SYSTEM FactoryioLuaJITDemo
  (* Version 1.0, 2021-07-28, Tuojian Lyu *)
  APPLICATION VariablesInitApp
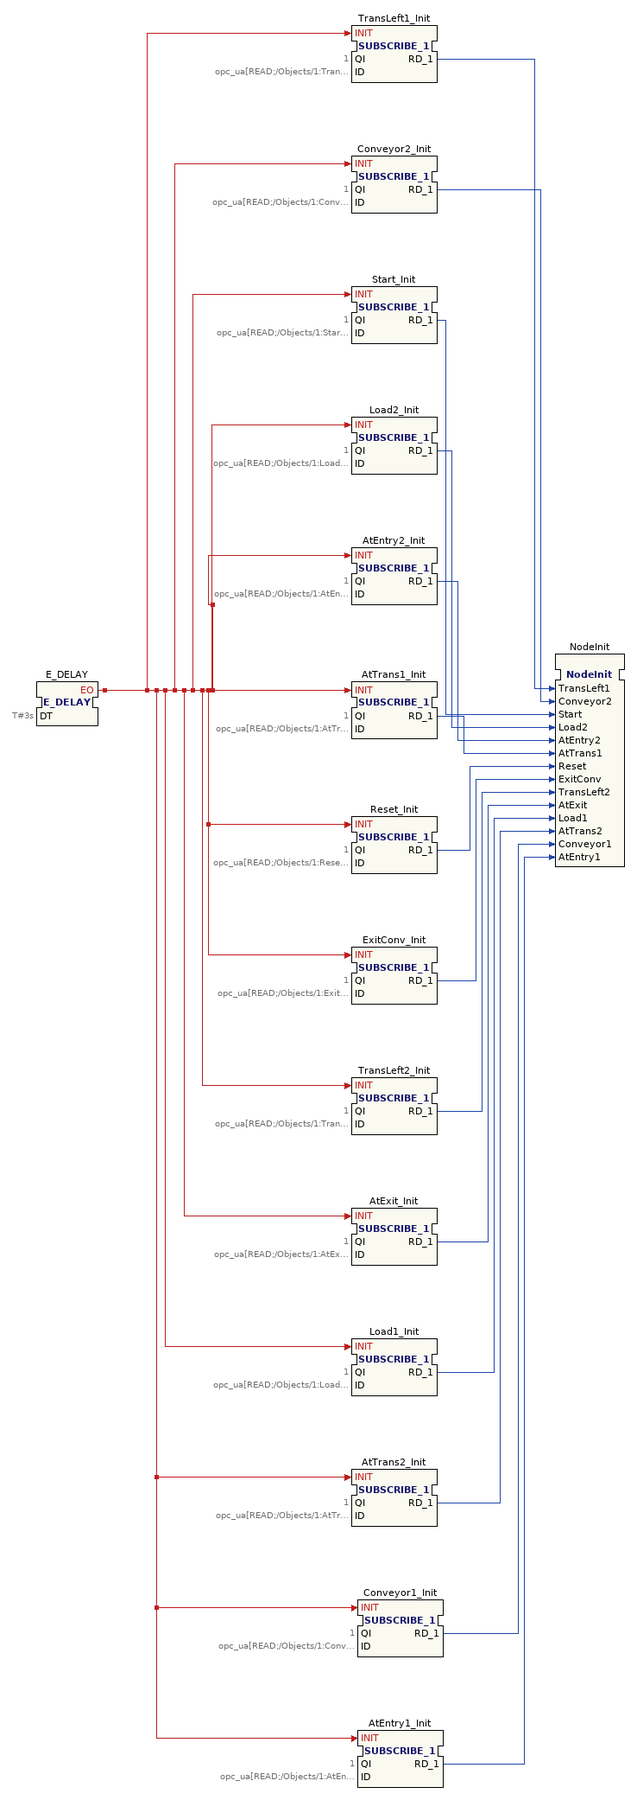
    FBS
      TransLeft1_Init : SUBSCRIBE_1(QI := 1, ID := opc_ua[READ;/Objects/1:TransLeft1]);
      Conveyor2_Init : SUBSCRIBE_1(QI := 1, ID := opc_ua[READ;/Objects/1:Conveyor2]);
      Start_Init : SUBSCRIBE_1(QI := 1, ID := opc_ua[READ;/Objects/1:Start]);
      AtEntry2_Init : SUBSCRIBE_1(QI := 1, ID := opc_ua[READ;/Objects/1:AtEntry2]);
      Load2_Init : SUBSCRIBE_1(QI := 1, ID := opc_ua[READ;/Objects/1:Load2]);
      Reset_Init : SUBSCRIBE_1(QI := 1, ID := opc_ua[READ;/Objects/1:Reset]);
      AtTrans1_Init : SUBSCRIBE_1(QI := 1, ID := opc_ua[READ;/Objects/1:AtTrans1]);
      TransLeft2_Init : SUBSCRIBE_1(QI := 1, ID := opc_ua[READ;/Objects/1:TransLeft2]);
      ExitConv_Init : SUBSCRIBE_1(QI := 1, ID := opc_ua[READ;/Objects/1:ExitConv]);
      Load1_Init : SUBSCRIBE_1(QI := 1, ID := opc_ua[READ;/Objects/1:Load1]);
      AtExit_Init : SUBSCRIBE_1(QI := 1, ID := opc_ua[READ;/Objects/1:AtExit]);
      AtTrans2_Init : SUBSCRIBE_1(QI := 1, ID := opc_ua[READ;/Objects/1:AtTrans2]);
      E_DELAY : E_DELAY(DT := T#3s);
      Conveyor1_Init : SUBSCRIBE_1(QI := 1, ID := opc_ua[READ;/Objects/1:Conveyor1]);
      AtEntry1_Init : SUBSCRIBE_1(QI := 1, ID := opc_ua[READ;/Objects/1:AtEntry1]);
      NodeInit : NodeInit;
    END_FBS
    EVENT_CONNECTIONS
      E_DELAY.EO TO TransLeft1_Init.INIT;
      E_DELAY.EO TO Conveyor2_Init.INIT;
      E_DELAY.EO TO Start_Init.INIT;
      E_DELAY.EO TO Load2_Init.INIT;
      E_DELAY.EO TO AtEntry2_Init.INIT;
      E_DELAY.EO TO AtTrans1_Init.INIT;
      E_DELAY.EO TO Reset_Init.INIT;
      E_DELAY.EO TO ExitConv_Init.INIT;
      E_DELAY.EO TO TransLeft2_Init.INIT;
      E_DELAY.EO TO AtExit_Init.INIT;
      E_DELAY.EO TO Load1_Init.INIT;
      E_DELAY.EO TO AtTrans2_Init.INIT;
      E_DELAY.EO TO Conveyor1_Init.INIT;
      E_DELAY.EO TO AtEntry1_Init.INIT;
    END_CONNECTIONS
    DATA_CONNECTIONS
      TransLeft1_Init.RD_1 TO NodeInit.TransLeft1;
      Conveyor2_Init.RD_1 TO NodeInit.Conveyor2;
      Start_Init.RD_1 TO NodeInit.Start;
      Load2_Init.RD_1 TO NodeInit.Load2;
      AtEntry2_Init.RD_1 TO NodeInit.AtEntry2;
      AtTrans1_Init.RD_1 TO NodeInit.AtTrans1;
      Reset_Init.RD_1 TO NodeInit.Reset;
      ExitConv_Init.RD_1 TO NodeInit.ExitConv;
      TransLeft2_Init.RD_1 TO NodeInit.TransLeft2;
      AtExit_Init.RD_1 TO NodeInit.AtExit;
      Load1_Init.RD_1 TO NodeInit.Load1;
      AtTrans2_Init.RD_1 TO NodeInit.AtTrans2;
      Conveyor1_Init.RD_1 TO NodeInit.Conveyor1;
      AtEntry1_Init.RD_1 TO NodeInit.AtEntry1;
    END_CONNECTIONS
  END_APPLICATION
  APPLICATION FactoryioLuaJITDemo
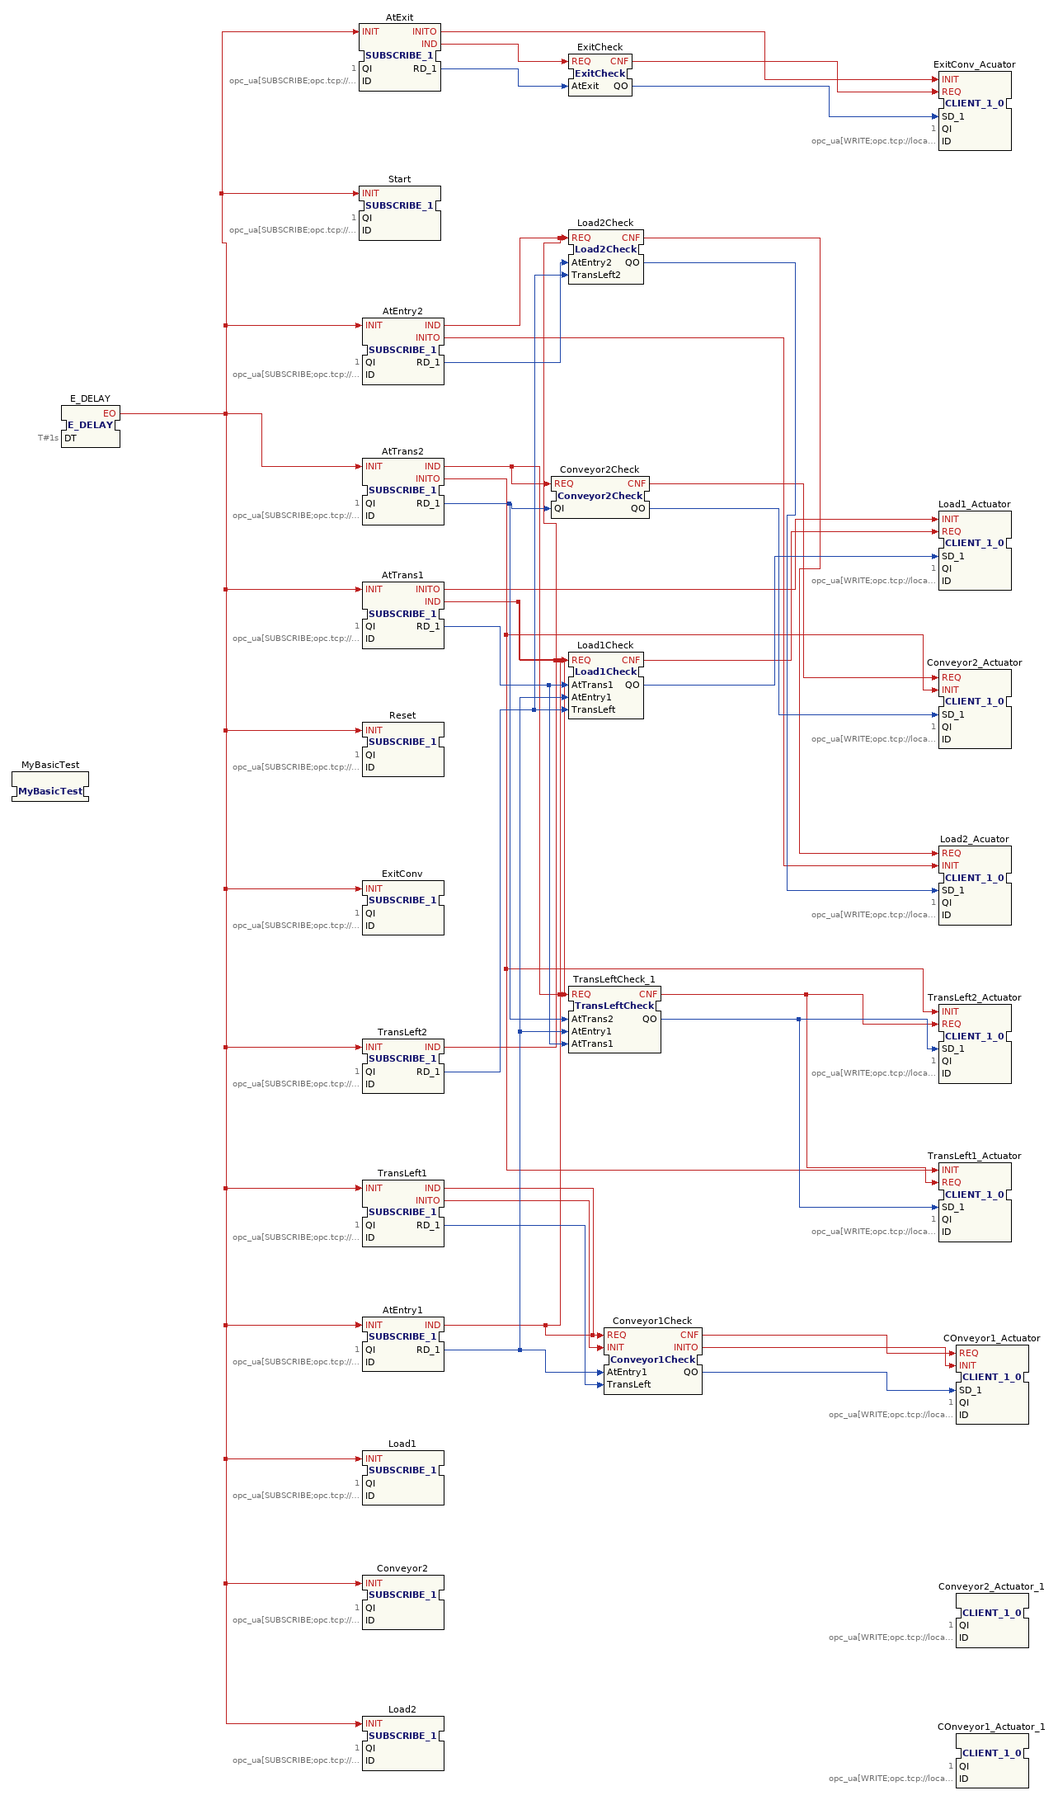
    FBS
      Load1_Actuator : CLIENT_1_0(QI := 1, ID := opc_ua[WRITE;opc.tcp://localhost:4840#;/Objects/1:Load1]);
      ExitConv_Acuator : CLIENT_1_0(QI := 1, ID := opc_ua[WRITE;opc.tcp://localhost:4840#;/Objects/1:ExitConv]);
      Start : SUBSCRIBE_1(QI := 1, ID := opc_ua[SUBSCRIBE;opc.tcp://localhost:4840#;/Objects/1:Start]);
      AtExit : SUBSCRIBE_1(QI := 1, ID := opc_ua[SUBSCRIBE;opc.tcp://localhost:4840#;/Objects/1:AtExit]);
      TransLeft1_Actuator : CLIENT_1_0(QI := 1, ID := opc_ua[WRITE;opc.tcp://localhost:4840#;/Objects/1:TransLeft1]);
      TransLeft2_Actuator : CLIENT_1_0(QI := 1, ID := opc_ua[WRITE;opc.tcp://localhost:4840#;/Objects/1:TransLeft2]);
      AtTrans2 : SUBSCRIBE_1(QI := 1, ID := opc_ua[SUBSCRIBE;opc.tcp://localhost:4840#;/Objects/1:AtTrans2]);
      Conveyor2_Actuator : CLIENT_1_0(QI := 1, ID := opc_ua[WRITE;opc.tcp://localhost:4840#;/Objects/1:Conveyor2]);
      AtEntry2 : SUBSCRIBE_1(QI := 1, ID := opc_ua[SUBSCRIBE;opc.tcp://localhost:4840#;/Objects/1:AtEntry2]);
      AtTrans1 : SUBSCRIBE_1(QI := 1, ID := opc_ua[SUBSCRIBE;opc.tcp://localhost:4840#;/Objects/1:AtTrans1]);
      E_DELAY : E_DELAY(DT := T#1s);
      ExitConv : SUBSCRIBE_1(QI := 1, ID := opc_ua[SUBSCRIBE;opc.tcp://localhost:4840#;/Objects/1:ExitConv]);
      Conveyor2 : SUBSCRIBE_1(QI := 1, ID := opc_ua[SUBSCRIBE;opc.tcp://localhost:4840#;/Objects/1:Conveyor2]);
      TransLeft2 : SUBSCRIBE_1(QI := 1, ID := opc_ua[SUBSCRIBE;opc.tcp://localhost:4840#;/Objects/1:TransLeft2]);
      Load1 : SUBSCRIBE_1(QI := 1, ID := opc_ua[SUBSCRIBE;opc.tcp://localhost:4840#;/Objects/1:Load1]);
      TransLeft1 : SUBSCRIBE_1(QI := 1, ID := opc_ua[SUBSCRIBE;opc.tcp://localhost:4840#;/Objects/1:TransLeft1]);
      Load2 : SUBSCRIBE_1(QI := 1, ID := opc_ua[SUBSCRIBE;opc.tcp://localhost:4840#;/Objects/1:Load2]);
      Reset : SUBSCRIBE_1(QI := 1, ID := opc_ua[SUBSCRIBE;opc.tcp://localhost:4840#;/Objects/1:Reset]);
      Load2_Acuator : CLIENT_1_0(QI := 1, ID := opc_ua[WRITE;opc.tcp://localhost:4840#;/Objects/1:Load2]);
      Conveyor2Check : Conveyor2Check;
      Load2Check : Load2Check;
      ExitCheck : ExitCheck;
      COnveyor1_Actuator : CLIENT_1_0(QI := 1, ID := opc_ua[WRITE;opc.tcp://localhost:4840#;/Objects/1:Conveyor1]);
      AtEntry1 : SUBSCRIBE_1(QI := 1, ID := opc_ua[SUBSCRIBE;opc.tcp://localhost:4840#;/Objects/1:AtEntry1]);
      Load1Check : Load1Check;
      Conveyor1Check : Conveyor1Check;
      TransLeftCheck_1 : TransLeftCheck;
      COnveyor1_Actuator_1 : CLIENT_1_0(QI := 1, ID := opc_ua[WRITE;opc.tcp://localhost:4840#;/Objects/1:Conveyor1]);
      Conveyor2_Actuator_1 : CLIENT_1_0(QI := 1, ID := opc_ua[WRITE;opc.tcp://localhost:4840#;/Objects/1:Conveyor2]);
      MyBasicTest : MyBasicTest;
    END_FBS
    EVENT_CONNECTIONS
      E_DELAY.EO TO AtExit.INIT;
      E_DELAY.EO TO Start.INIT;
      E_DELAY.EO TO AtEntry2.INIT;
      E_DELAY.EO TO AtTrans2.INIT;
      E_DELAY.EO TO AtTrans1.INIT;
      E_DELAY.EO TO TransLeft1.INIT;
      E_DELAY.EO TO ExitConv.INIT;
      E_DELAY.EO TO Load1.INIT;
      E_DELAY.EO TO Conveyor2.INIT;
      E_DELAY.EO TO TransLeft2.INIT;
      E_DELAY.EO TO Load2.INIT;
      E_DELAY.EO TO Reset.INIT;
      Conveyor2Check.CNF TO Conveyor2_Actuator.REQ;
      AtTrans2.IND TO Conveyor2Check.REQ;
      AtEntry2.IND TO Load2Check.REQ;
      Load2Check.CNF TO Load2_Acuator.REQ;
      AtTrans2.INITO TO Conveyor2_Actuator.INIT;
      AtEntry2.INITO TO Load2_Acuator.INIT;
      AtTrans2.INITO TO TransLeft2_Actuator.INIT;
      AtTrans2.INITO TO TransLeft1_Actuator.INIT;
      AtTrans1.INITO TO Load1_Actuator.INIT;
      AtExit.INITO TO ExitConv_Acuator.INIT;
      AtExit.IND TO ExitCheck.REQ;
      ExitCheck.CNF TO ExitConv_Acuator.REQ;
      E_DELAY.EO TO AtEntry1.INIT;
      AtTrans1.IND TO Load1Check.REQ;
      AtEntry1.IND TO Load1Check.REQ;
      TransLeft2.IND TO Load1Check.REQ;
      Load1Check.CNF TO Load1_Actuator.REQ;
      TransLeft2.IND TO Load2Check.REQ;
      AtEntry1.IND TO Conveyor1Check.REQ;
      TransLeft1.IND TO Conveyor1Check.REQ;
      Conveyor1Check.CNF TO COnveyor1_Actuator.REQ;
      TransLeft1.INITO TO Conveyor1Check.INIT;
      Conveyor1Check.INITO TO COnveyor1_Actuator.INIT;
      AtTrans2.IND TO TransLeftCheck_1.REQ;
      AtEntry1.IND TO TransLeftCheck_1.REQ;
      AtTrans1.IND TO TransLeftCheck_1.REQ;
      TransLeftCheck_1.CNF TO TransLeft2_Actuator.REQ;
      TransLeftCheck_1.CNF TO TransLeft1_Actuator.REQ;
    END_CONNECTIONS
    DATA_CONNECTIONS
      Conveyor2Check.QO TO Conveyor2_Actuator.SD_1;
      AtTrans2.RD_1 TO Conveyor2Check.QI;
      AtEntry2.RD_1 TO Load2Check.AtEntry2;
      TransLeft2.RD_1 TO Load2Check.TransLeft2;
      Load2Check.QO TO Load2_Acuator.SD_1;
      AtExit.RD_1 TO ExitCheck.AtExit;
      ExitCheck.QO TO ExitConv_Acuator.SD_1;
      AtTrans1.RD_1 TO Load1Check.AtTrans1;
      AtEntry1.RD_1 TO Load1Check.AtEntry1;
      TransLeft2.RD_1 TO Load1Check.TransLeft;
      Load1Check.QO TO Load1_Actuator.SD_1;
      AtEntry1.RD_1 TO Conveyor1Check.AtEntry1;
      TransLeft1.RD_1 TO Conveyor1Check.TransLeft;
      Conveyor1Check.QO TO COnveyor1_Actuator.SD_1;
      AtTrans2.RD_1 TO TransLeftCheck_1.AtTrans2;
      AtEntry1.RD_1 TO TransLeftCheck_1.AtEntry1;
      AtTrans1.RD_1 TO TransLeftCheck_1.AtTrans1;
      TransLeftCheck_1.QO TO TransLeft2_Actuator.SD_1;
      TransLeftCheck_1.QO TO TransLeft1_Actuator.SD_1;
    END_CONNECTIONS
  END_APPLICATION
  DEVICE FORTE_PC : FORTE_PC(MGR_ID := "localhost:61499")
    {SET_ATTRIBUTE(Profile, DynamicTypeLoad)} (* device profile *)
    {SET_ATTRIBUTE(FBType, GEN_E_MUX, F_LT, F_LWORD_TO_WORD, F_TAN, F_DINT_TO_UINT, F_BYTE_TO_DINT, F_ADD_DT_TIME, F_TIME_IN_US_TO_LREAL, F_INT_TO_UDINT, F_ADD_TOD_TIME, F_SUB_DT_DT, F_DT_TO_TOD, F_WSTRING_TO_REAL, F_UINT_TO_BCD_WORD, F_UDINT_TO_REAL, F_REAL_TO_UDINT, F_DWORD_TO_WORD, F_MUL, FB_CTUD_LINT, TEST_CONDITION, F_LE, GEN_SUBSCRIBE, F_LN, FB_CTD_DINT, GEN_OR, E_CYCLE, FB_F_TRIG, F_LREAL_TO_SINT, E_F_TRIG, F_LWORD_TO_UINT, E_RS, F_UINT_TO_WORD, F_WORD_TO_DINT, F_OR, F_WORD_TO_BYTE, F_TIME_IN_NS_TO_ULINT, FB_CTD_ULINT, FB_TOF, STEST_END, F_NE, FB_TON, F_STRING_TO_UINT, F_LWORD_TO_ULINT, F_INT_TO_STRING, F_INT_TO_BYTE, F_INT_TO_DINT, F_ULINT_TO_LINT, F_DWORD_TO_UINT, F_WSTRING_TO_ULINT, F_WSTRING_TO_LWORD, F_STRING_TO_DWORD, DWORD2DWORD, F_TIME_IN_NS_TO_LINT, F_DINT_TO_WSTRING, E_SELECT, F_LINT_TO_STRING, FB_CTUD, F_MULTIME, F_USINT_TO_INT, LocalizedText2LocalizedText, NodeInit, F_DWORD_TO_UDINT, F_UINT_TO_LWORD, F_SINT_TO_LWORD, GEN_F_MUX, USINT2USINT, F_LINT_TO_SINT, F_WORD_TO_USINT, F_DWORD_TO_INT, F_LREAL_TO_REAL, F_BOOL_TO_LINT, F_LEFT, FB_CTD, E_SR, F_UDINT_TO_BCD_DWORD, GEN_XOR, F_DINT_TO_WORD, F_SUB_TOD_TIME, E_RESTART, E_PERMIT, TIME2TIME, F_UINT_TO_SINT, F_XOR, F_STRING_TO_WORD, F_SEL, F_ULINT_TO_LREAL, F_SINT_TO_LREAL, F_DINT_TO_SINT, E_TimeOut, F_BYTE_TO_UDINT, F_REPLACE, F_LINT_TO_USINT, F_ABS, F_WORD_TO_LWORD, E_DELAY, GEN_ADD, F_INT_TO_WSTRING, F_STRING_TO_ULINT, F_USINT_TO_STRING, F_DINT_TO_USINT, F_STRING_TO_BOOL, F_DWORD_TO_WSTRING, F_INT_TO_REAL, F_DWORD_TO_STRING, E_CTU, F_TIME_TO_STRING, F_WSTRING_TO_BYTE, F_USINT_TO_WSTRING, F_WSTRING_TO_DINT, F_WSTRING_TO_DWORD, F_MOVE, F_WSTRING_TO_STRING, F_USINT_TO_LINT, F_DIV, F_WSTRING_TO_SINT, E_CTD, F_UINT_TO_DWORD, F_LWORD_TO_LINT, F_STRING_TO_TIME, FB_CTUD_DINT, F_ADD, F_BYTE_TO_LINT, F_TIME_IN_MS_TO_LREAL, F_LREAL_TO_UINT, F_ACOS, F_DWORD_TO_LINT, F_SHL, F_REAL_TO_ULINT, F_ULINT_TO_UINT, F_UDINT_TO_SINT, F_SHR, F_BOOL_TO_INT, UINT2UINT, F_WORD_TO_DWORD, F_INT_TO_LWORD, F_USINT_TO_UINT, F_LREAL_TO_WSTRING, F_INT_TO_ULINT, GEN_CSV_WRITER, F_LINT_TO_WORD, F_UINT_TO_LREAL, F_STRING_TO_SINT, F_SINT_TO_WORD, F_STRING_TO_WSTRING, STRING2STRING, F_LREAL_TO_DINT, F_SIN, F_UINT_TO_USINT, FB_CTU_LINT, F_DINT_TO_ULINT, F_REAL_TO_UINT, RMT_RES, F_ULINT_TO_WORD, F_INT_TO_LINT, E_D_FF, F_STRING_TO_USINT, FB_CTD_LINT, FB_R_TRIG, F_INT_TO_DWORD, F_WORD_TO_LINT, F_UDINT_TO_INT, REAL2REAL, F_LREAL_TO_STRING, F_WSTRING_TO_INT, F_LREAL_TO_USINT, F_DINT_TO_LWORD, DEV_MGR, F_SINT_TO_UINT, E_CTUD, E_RDELAY, F_SINT_TO_ULINT, F_LINT_TO_ULINT, F_RIGHT, F_SINT_TO_INT, F_LWORD_TO_WSTRING, SINT2SINT, FB_CTD_UDINT, F_LINT_TO_LWORD, F_LWORD_TO_UDINT, F_LWORD_TO_STRING, F_TRUNC, F_ULINT_TO_DWORD, F_TIME_IN_S_TO_LREAL, F_BOOL_TO_DWORD, E_TRAIN, OUT_ANY_CONSOLE, F_ULINT_TO_SINT, F_DINT_TO_LINT, F_BOOL_TO_USINT, F_UDINT_TO_DWORD, GEN_E_DEMUX, F_SQRT, F_BOOL_TO_DINT, F_BOOL_TO_BYTE, F_UINT_TO_INT, F_TIME_IN_S_TO_LINT, F_ULINT_TO_USINT, F_UINT_TO_REAL, F_LREAL_TO_LWORD, F_SINT_TO_LINT, F_MAX, F_LREAL_TO_INT, F_UDINT_TO_LWORD, INT2INT, F_BYTE_TO_ULINT, F_UDINT_TO_WORD, F_LINT_TO_UINT, F_TIME_IN_US_TO_ULINT, F_COS, F_TIME_IN_NS_TO_LREAL, F_REAL_TO_LINT, F_STRING_TO_LWORD, F_BYTE_TO_STRING, F_USINT_TO_WORD, E_REND, F_ASIN, F_REAL_TO_INT, F_BOOL_TO_LWORD, F_WORD_BCD_TO_UINT, F_BOOL_TO_SINT, F_BYTE_TO_INT, F_BOOL_TO_ULINT, EMB_RES, F_BYTE_TO_WORD, F_STRING_TO_INT, F_USINT_TO_LWORD, F_DWORD_TO_DINT, F_ULINT_TO_LWORD, GEN_APPEND_STRING, F_USINT_TO_ULINT, GEN_SUBL, F_DWORD_TO_BYTE, F_DIVTIME, F_ROL, F_LWORD_TO_DINT, F_WORD_TO_SINT, F_STRING_TO_REAL, F_LWORD_TO_BYTE, FB_CTU_DINT, GEN_AND, F_AND, F_ROR, GEN_CLIENT, F_ULINT_TO_WSTRING, F_SINT_TO_STRING, F_LREAL_TO_LINT, WSTRING2WSTRING, F_WORD_TO_INT, F_UINT_TO_BYTE, F_UDINT_TO_UINT, F_SINT_TO_UDINT, F_UINT_TO_DINT, F_UINT_TO_UDINT, F_UINT_TO_WSTRING, F_WSTRING_TO_UINT, F_DINT_TO_UDINT, E_SPLIT, F_DWORD_TO_LWORD, F_USINT_TO_SINT, F_ULINT_TO_BCD_LWORD, F_BYTE_BCD_TO_USINT, F_DWORD_TO_ULINT, F_BYTE_TO_SINT, F_BYTE_TO_WSTRING, GEN_ARRAY2ARRAY, F_DT_TO_DATE, GEN_STRUCT_DEMUX, F_LEN, GEN_STRUCT_MUX, F_INT_TO_WORD, FB_RANDOM, F_LINT_TO_UDINT, F_EXP, F_USINT_TO_DWORD, F_TIME_IN_MS_TO_ULINT, F_REAL_TO_SINT, F_INT_TO_USINT, F_UDINT_TO_WSTRING, F_EXPT, F_SUB, F_ULINT_TO_REAL, F_REAL_TO_LREAL, F_MID, F_BYTE_TO_UINT, F_BYTE_TO_DWORD, F_INT_TO_UINT, F_DWORD_TO_REAL, F_DINT_TO_BYTE, F_WORD_TO_STRING, F_REAL_TO_STRING, F_SUB_TOD_TOD, SET_AT_INDEX, F_MIN, F_LREAL_TO_ULINT, F_STRING_TO_BYTE, F_BYTE_TO_LWORD, F_STRING_TO_DINT, F_WORD_TO_WSTRING, BOOL2BOOL, F_LINT_TO_INT, F_WSTRING_TO_TIME, FB_CTU_UDINT, F_WSTRING_TO_BOOL, F_INSERT, F_SUB_DT_TIME, F_FIND, F_UDINT_TO_ULINT, F_WORD_TO_UDINT, F_DINT_TO_DWORD, F_WSTRING_TO_USINT, GEN_VALUES2ARRAY, GEN_ARRAY2VALUES, F_WSTRING_TO_WORD, F_DINT_TO_STRING, F_WORD_TO_UINT, F_TIME_IN_US_TO_LINT, F_LINT_TO_DWORD, F_CONCAT, FB_CTUD_ULINT, F_UDINT_TO_LINT, F_SUB_DATE_DATE, F_LWORD_TO_LREAL, F_LWORD_TO_INT, WORD2WORD, E_STOPWATCH, F_LIMIT, F_TIME_IN_S_TO_ULINT, F_LWORD_TO_USINT, F_REAL_TO_DINT, F_DWORD_TO_USINT, E_MERGE, F_SINT_TO_DWORD, E_DEMUX, F_BOOL_TO_UDINT, BYTE2BYTE, FB_TP, F_USINT_TO_BCD_BYTE, F_SINT_TO_DINT, F_UINT_TO_LINT, F_SINT_TO_BYTE, F_ATAN, F_LINT_TO_BYTE, F_BYTE_TO_USINT, F_ULINT_TO_UDINT, FB_SR, F_NOT, F_DINT_TO_INT, F_LINT_TO_DINT, F_DELETE, FB_CTU, GEN_SERVER, GEN_PUBL, F_UDINT_TO_LREAL, F_BOOL_TO_UINT, F_UINT_TO_STRING, E_R_TRIG, F_GE, F_LWORD_BCD_TO_ULINT, F_UDINT_TO_STRING, F_REAL_TO_WSTRING, FB_RS, F_MUX_2, F_LINT_TO_WSTRING, F_USINT_TO_UDINT, F_UINT_TO_ULINT, F_EQ, E_T_FF, F_USINT_TO_REAL, LREAL2LREAL, F_STRING_TO_LREAL, F_ULINT_TO_STRING, F_MOD, E_RTimeOut, F_ULINT_TO_DINT, F_ULINT_TO_BYTE, F_WSTRING_TO_UDINT, F_TIME_TO_WSTRING, GET_STRUCT_VALUE, GEN_PUBLISH, F_REAL_TO_DWORD, F_DWORD_BCD_TO_UDINT, F_INT_TO_LREAL, F_SINT_TO_WSTRING, F_LWORD_TO_SINT, F_GT, F_LINT_TO_REAL, F_TIME_IN_MS_TO_LINT, F_SINT_TO_REAL, F_LOG, F_ULINT_TO_INT, F_DWORD_TO_SINT, F_BOOL_TO_WORD, F_REAL_TO_USINT, E_SWITCH, F_LINT_TO_LREAL, F_STRING_TO_LINT, F_SINT_TO_USINT, F_DINT_TO_REAL, DINT2DINT, F_WORD_TO_ULINT, F_INT_TO_SINT, F_CONCAT_DATE_TOD, F_WSTRING_TO_LREAL, GET_AT_INDEX, F_USINT_TO_LREAL, F_BOOL_TO_WSTRING, FB_CTU_ULINT, F_DINT_TO_LREAL, UDINT2UDINT, F_USINT_TO_BYTE, F_BOOL_TO_STRING, F_LWORD_TO_DWORD, F_LREAL_TO_UDINT, F_STRING_TO_UDINT, F_UDINT_TO_DINT, F_UDINT_TO_BYTE, F_WSTRING_TO_LINT, F_USINT_TO_DINT)} (* created during deployment *)
    RESOURCE EMB_RES : EMB_RES
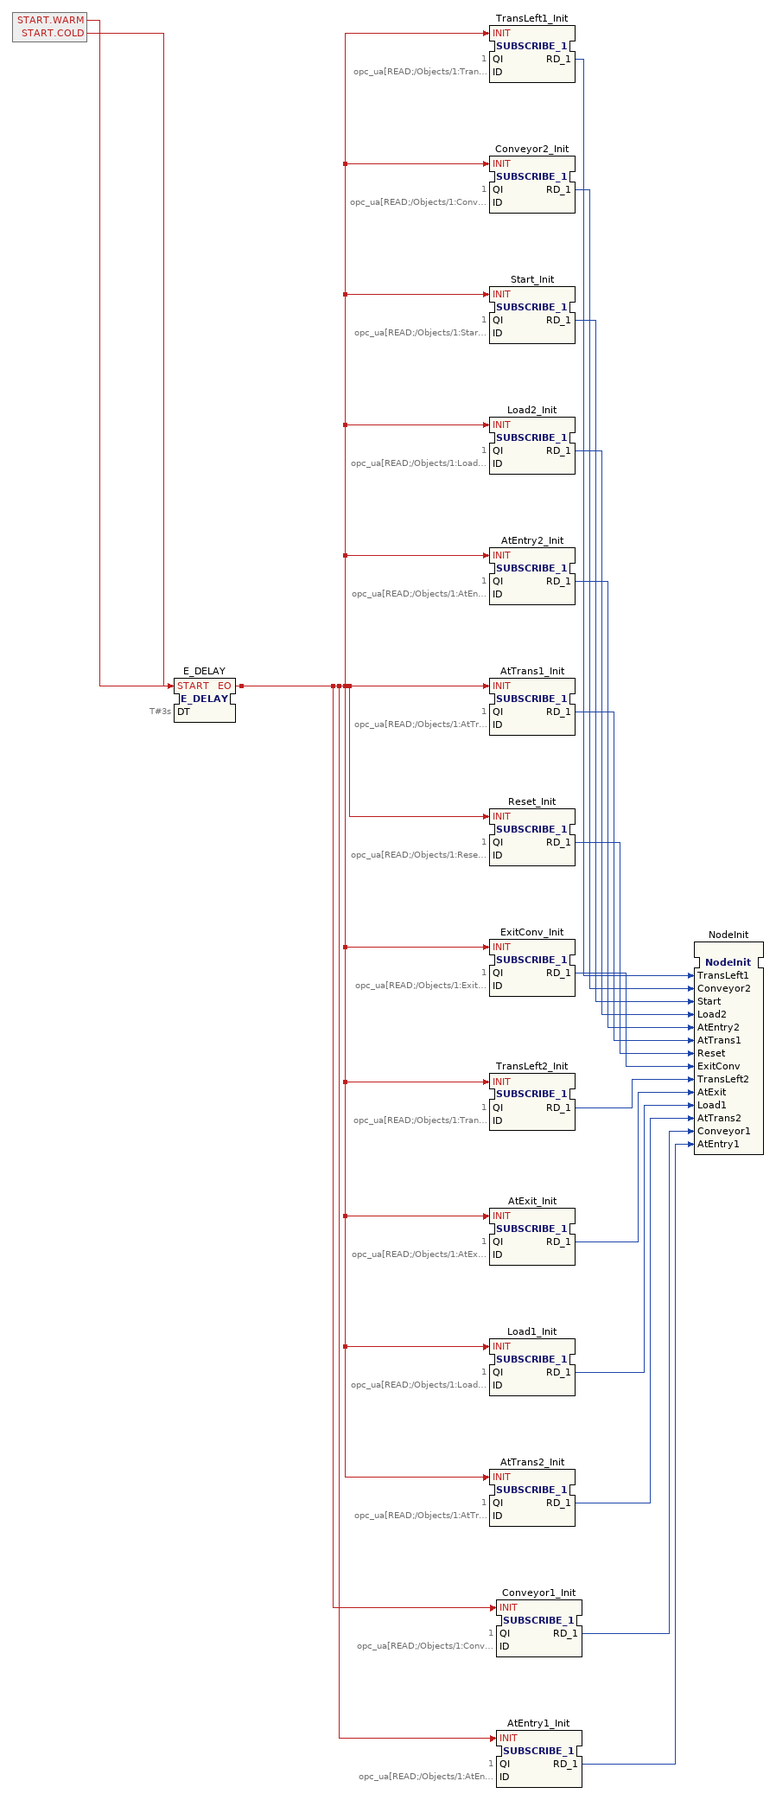
      FBS
        E_DELAY : E_DELAY(DT := T#3s);
        AtTrans2_Init : SUBSCRIBE_1(QI := 1, ID := opc_ua[READ;/Objects/1:AtTrans2]);
        AtExit_Init : SUBSCRIBE_1(QI := 1, ID := opc_ua[READ;/Objects/1:AtExit]);
        Load1_Init : SUBSCRIBE_1(QI := 1, ID := opc_ua[READ;/Objects/1:Load1]);
        ExitConv_Init : SUBSCRIBE_1(QI := 1, ID := opc_ua[READ;/Objects/1:ExitConv]);
        TransLeft2_Init : SUBSCRIBE_1(QI := 1, ID := opc_ua[READ;/Objects/1:TransLeft2]);
        AtTrans1_Init : SUBSCRIBE_1(QI := 1, ID := opc_ua[READ;/Objects/1:AtTrans1]);
        Reset_Init : SUBSCRIBE_1(QI := 1, ID := opc_ua[READ;/Objects/1:Reset]);
        Load2_Init : SUBSCRIBE_1(QI := 1, ID := opc_ua[READ;/Objects/1:Load2]);
        AtEntry2_Init : SUBSCRIBE_1(QI := 1, ID := opc_ua[READ;/Objects/1:AtEntry2]);
        Start_Init : SUBSCRIBE_1(QI := 1, ID := opc_ua[READ;/Objects/1:Start]);
        Conveyor2_Init : SUBSCRIBE_1(QI := 1, ID := opc_ua[READ;/Objects/1:Conveyor2]);
        TransLeft1_Init : SUBSCRIBE_1(QI := 1, ID := opc_ua[READ;/Objects/1:TransLeft1]);
        Conveyor1_Init : SUBSCRIBE_1(QI := 1, ID := opc_ua[READ;/Objects/1:Conveyor1]);
        AtEntry1_Init : SUBSCRIBE_1(QI := 1, ID := opc_ua[READ;/Objects/1:AtEntry1]);
        NodeInit : NodeInit;
      END_FBS
      EVENT_CONNECTIONS
        START.WARM TO E_DELAY.START;
        START.COLD TO E_DELAY.START;
        E_DELAY.EO TO AtTrans2_Init.INIT;
        E_DELAY.EO TO AtExit_Init.INIT;
        E_DELAY.EO TO Load1_Init.INIT;
        E_DELAY.EO TO ExitConv_Init.INIT;
        E_DELAY.EO TO TransLeft2_Init.INIT;
        E_DELAY.EO TO AtTrans1_Init.INIT;
        E_DELAY.EO TO Reset_Init.INIT;
        E_DELAY.EO TO Load2_Init.INIT;
        E_DELAY.EO TO AtEntry2_Init.INIT;
        E_DELAY.EO TO Start_Init.INIT;
        E_DELAY.EO TO Conveyor2_Init.INIT;
        E_DELAY.EO TO TransLeft1_Init.INIT;
        E_DELAY.EO TO Conveyor1_Init.INIT;
        E_DELAY.EO TO AtEntry1_Init.INIT;
      END_CONNECTIONS
      DATA_CONNECTIONS
        TransLeft1_Init.RD_1 TO NodeInit.TransLeft1;
        Conveyor2_Init.RD_1 TO NodeInit.Conveyor2;
        Start_Init.RD_1 TO NodeInit.Start;
        Load2_Init.RD_1 TO NodeInit.Load2;
        AtEntry2_Init.RD_1 TO NodeInit.AtEntry2;
        AtTrans1_Init.RD_1 TO NodeInit.AtTrans1;
        Reset_Init.RD_1 TO NodeInit.Reset;
        ExitConv_Init.RD_1 TO NodeInit.ExitConv;
        TransLeft2_Init.RD_1 TO NodeInit.TransLeft2;
        AtExit_Init.RD_1 TO NodeInit.AtExit;
        Load1_Init.RD_1 TO NodeInit.Load1;
        AtTrans2_Init.RD_1 TO NodeInit.AtTrans2;
        Conveyor1_Init.RD_1 TO NodeInit.Conveyor1;
        AtEntry1_Init.RD_1 TO NodeInit.AtEntry1;
      END_CONNECTIONS
    END_RESOURCE
  END_DEVICE
  DEVICE FORTE_PC_1 : FORTE_PC(MGR_ID := "localhost:61500")
    {SET_ATTRIBUTE(Profile, DynamicTypeLoad)} (* device profile *)
    {SET_ATTRIBUTE(FBType, GEN_E_MUX, F_LT, F_LWORD_TO_WORD, F_TAN, F_DINT_TO_UINT, F_BYTE_TO_DINT, F_ADD_DT_TIME, F_TIME_IN_US_TO_LREAL, F_INT_TO_UDINT, F_ADD_TOD_TIME, F_SUB_DT_DT, F_DT_TO_TOD, F_WSTRING_TO_REAL, F_UINT_TO_BCD_WORD, F_UDINT_TO_REAL, F_REAL_TO_UDINT, F_DWORD_TO_WORD, F_MUL, FB_CTUD_LINT, TEST_CONDITION, F_LE, GEN_SUBSCRIBE, F_LN, FB_CTD_DINT, GEN_OR, E_CYCLE, FB_F_TRIG, F_LREAL_TO_SINT, E_F_TRIG, F_LWORD_TO_UINT, E_RS, F_UINT_TO_WORD, F_WORD_TO_DINT, F_OR, F_WORD_TO_BYTE, F_TIME_IN_NS_TO_ULINT, FB_CTD_ULINT, FB_TOF, STEST_END, F_NE, FB_TON, F_STRING_TO_UINT, F_LWORD_TO_ULINT, F_INT_TO_STRING, F_INT_TO_BYTE, F_INT_TO_DINT, F_ULINT_TO_LINT, F_DWORD_TO_UINT, F_WSTRING_TO_ULINT, F_WSTRING_TO_LWORD, F_STRING_TO_DWORD, DWORD2DWORD, F_TIME_IN_NS_TO_LINT, F_DINT_TO_WSTRING, E_SELECT, F_LINT_TO_STRING, FB_CTUD, F_MULTIME, F_USINT_TO_INT, LocalizedText2LocalizedText, F_DWORD_TO_UDINT, F_UINT_TO_LWORD, F_SINT_TO_LWORD, GEN_F_MUX, USINT2USINT, F_LINT_TO_SINT, F_WORD_TO_USINT, F_DWORD_TO_INT, F_LREAL_TO_REAL, F_BOOL_TO_LINT, F_LEFT, FB_CTD, E_SR, F_UDINT_TO_BCD_DWORD, GEN_XOR, F_DINT_TO_WORD, F_SUB_TOD_TIME, E_RESTART, E_PERMIT, TIME2TIME, F_UINT_TO_SINT, F_XOR, F_STRING_TO_WORD, F_SEL, F_ULINT_TO_LREAL, F_SINT_TO_LREAL, F_DINT_TO_SINT, E_TimeOut, F_BYTE_TO_UDINT, F_REPLACE, F_LINT_TO_USINT, F_ABS, F_WORD_TO_LWORD, MyBasicTest, E_DELAY, GEN_ADD, F_INT_TO_WSTRING, F_STRING_TO_ULINT, F_USINT_TO_STRING, F_DINT_TO_USINT, F_STRING_TO_BOOL, F_DWORD_TO_WSTRING, F_INT_TO_REAL, F_DWORD_TO_STRING, E_CTU, F_TIME_TO_STRING, F_WSTRING_TO_BYTE, F_USINT_TO_WSTRING, F_WSTRING_TO_DINT, F_WSTRING_TO_DWORD, F_MOVE, F_WSTRING_TO_STRING, F_USINT_TO_LINT, F_DIV, F_WSTRING_TO_SINT, E_CTD, F_UINT_TO_DWORD, F_LWORD_TO_LINT, F_STRING_TO_TIME, FB_CTUD_DINT, F_ADD, F_BYTE_TO_LINT, F_TIME_IN_MS_TO_LREAL, F_LREAL_TO_UINT, F_ACOS, F_DWORD_TO_LINT, F_SHL, F_REAL_TO_ULINT, F_ULINT_TO_UINT, F_UDINT_TO_SINT, F_SHR, F_BOOL_TO_INT, UINT2UINT, F_WORD_TO_DWORD, F_INT_TO_LWORD, F_USINT_TO_UINT, F_LREAL_TO_WSTRING, F_INT_TO_ULINT, GEN_CSV_WRITER, F_LINT_TO_WORD, F_UINT_TO_LREAL, F_STRING_TO_SINT, F_SINT_TO_WORD, F_STRING_TO_WSTRING, STRING2STRING, F_LREAL_TO_DINT, F_SIN, F_UINT_TO_USINT, FB_CTU_LINT, F_DINT_TO_ULINT, F_REAL_TO_UINT, RMT_RES, F_ULINT_TO_WORD, F_INT_TO_LINT, E_D_FF, F_STRING_TO_USINT, FB_CTD_LINT, FB_R_TRIG, F_INT_TO_DWORD, F_WORD_TO_LINT, F_UDINT_TO_INT, REAL2REAL, F_LREAL_TO_STRING, F_WSTRING_TO_INT, F_LREAL_TO_USINT, F_DINT_TO_LWORD, DEV_MGR, F_SINT_TO_UINT, E_CTUD, E_RDELAY, F_SINT_TO_ULINT, F_LINT_TO_ULINT, F_RIGHT, F_SINT_TO_INT, F_LWORD_TO_WSTRING, SINT2SINT, FB_CTD_UDINT, F_LINT_TO_LWORD, F_LWORD_TO_UDINT, F_LWORD_TO_STRING, F_TRUNC, F_ULINT_TO_DWORD, F_TIME_IN_S_TO_LREAL, F_BOOL_TO_DWORD, E_TRAIN, OUT_ANY_CONSOLE, F_ULINT_TO_SINT, F_DINT_TO_LINT, F_BOOL_TO_USINT, F_UDINT_TO_DWORD, GEN_E_DEMUX, F_SQRT, F_BOOL_TO_DINT, F_BOOL_TO_BYTE, F_UINT_TO_INT, F_TIME_IN_S_TO_LINT, F_ULINT_TO_USINT, F_UINT_TO_REAL, F_LREAL_TO_LWORD, F_SINT_TO_LINT, F_MAX, F_LREAL_TO_INT, F_UDINT_TO_LWORD, INT2INT, F_BYTE_TO_ULINT, F_UDINT_TO_WORD, F_LINT_TO_UINT, F_TIME_IN_US_TO_ULINT, F_COS, Conveyor2Check, F_TIME_IN_NS_TO_LREAL, F_REAL_TO_LINT, F_STRING_TO_LWORD, F_BYTE_TO_STRING, F_USINT_TO_WORD, E_REND, F_ASIN, TransLeftCheck, F_REAL_TO_INT, F_BOOL_TO_LWORD, F_WORD_BCD_TO_UINT, F_BOOL_TO_SINT, F_BYTE_TO_INT, F_BOOL_TO_ULINT, EMB_RES, F_BYTE_TO_WORD, F_STRING_TO_INT, F_USINT_TO_LWORD, F_DWORD_TO_DINT, F_ULINT_TO_LWORD, GEN_APPEND_STRING, F_USINT_TO_ULINT, GEN_SUBL, F_DWORD_TO_BYTE, F_DIVTIME, ExitCheck, F_ROL, F_LWORD_TO_DINT, F_WORD_TO_SINT, F_STRING_TO_REAL, F_LWORD_TO_BYTE, FB_CTU_DINT, GEN_AND, F_AND, F_ROR, GEN_CLIENT, F_ULINT_TO_WSTRING, F_SINT_TO_STRING, F_LREAL_TO_LINT, WSTRING2WSTRING, F_WORD_TO_INT, F_UINT_TO_BYTE, F_UDINT_TO_UINT, F_SINT_TO_UDINT, F_UINT_TO_DINT, F_UINT_TO_UDINT, F_UINT_TO_WSTRING, F_WSTRING_TO_UINT, F_DINT_TO_UDINT, E_SPLIT, F_DWORD_TO_LWORD, F_USINT_TO_SINT, F_ULINT_TO_BCD_LWORD, F_BYTE_BCD_TO_USINT, F_DWORD_TO_ULINT, F_BYTE_TO_SINT, F_BYTE_TO_WSTRING, GEN_ARRAY2ARRAY, F_DT_TO_DATE, GEN_STRUCT_DEMUX, F_LEN, GEN_STRUCT_MUX, F_INT_TO_WORD, FB_RANDOM, F_LINT_TO_UDINT, F_EXP, F_USINT_TO_DWORD, F_TIME_IN_MS_TO_ULINT, F_REAL_TO_SINT, F_INT_TO_USINT, Load2Check, F_UDINT_TO_WSTRING, F_EXPT, F_SUB, F_ULINT_TO_REAL, F_REAL_TO_LREAL, F_MID, F_BYTE_TO_UINT, F_BYTE_TO_DWORD, F_INT_TO_UINT, F_DWORD_TO_REAL, F_DINT_TO_BYTE, F_WORD_TO_STRING, F_REAL_TO_STRING, F_SUB_TOD_TOD, SET_AT_INDEX, F_MIN, F_LREAL_TO_ULINT, F_STRING_TO_BYTE, F_BYTE_TO_LWORD, F_STRING_TO_DINT, F_WORD_TO_WSTRING, BOOL2BOOL, F_LINT_TO_INT, F_WSTRING_TO_TIME, FB_CTU_UDINT, F_WSTRING_TO_BOOL, F_INSERT, F_SUB_DT_TIME, F_FIND, F_UDINT_TO_ULINT, F_WORD_TO_UDINT, F_DINT_TO_DWORD, Load1Check, F_WSTRING_TO_USINT, GEN_VALUES2ARRAY, GEN_ARRAY2VALUES, F_WSTRING_TO_WORD, F_DINT_TO_STRING, F_WORD_TO_UINT, F_TIME_IN_US_TO_LINT, F_LINT_TO_DWORD, F_CONCAT, FB_CTUD_ULINT, F_UDINT_TO_LINT, F_SUB_DATE_DATE, F_LWORD_TO_LREAL, F_LWORD_TO_INT, WORD2WORD, E_STOPWATCH, F_LIMIT, F_TIME_IN_S_TO_ULINT, F_LWORD_TO_USINT, F_REAL_TO_DINT, F_DWORD_TO_USINT, E_MERGE, F_SINT_TO_DWORD, E_DEMUX, F_BOOL_TO_UDINT, BYTE2BYTE, FB_TP, F_USINT_TO_BCD_BYTE, F_SINT_TO_DINT, F_UINT_TO_LINT, F_SINT_TO_BYTE, F_ATAN, F_LINT_TO_BYTE, F_BYTE_TO_USINT, F_ULINT_TO_UDINT, FB_SR, F_NOT, F_DINT_TO_INT, F_LINT_TO_DINT, F_DELETE, FB_CTU, GEN_SERVER, GEN_PUBL, F_UDINT_TO_LREAL, F_BOOL_TO_UINT, F_UINT_TO_STRING, E_R_TRIG, F_GE, F_LWORD_BCD_TO_ULINT, F_UDINT_TO_STRING, F_REAL_TO_WSTRING, FB_RS, F_MUX_2, F_LINT_TO_WSTRING, F_USINT_TO_UDINT, F_UINT_TO_ULINT, F_EQ, E_T_FF, F_USINT_TO_REAL, LREAL2LREAL, F_STRING_TO_LREAL, F_ULINT_TO_STRING, F_MOD, E_RTimeOut, F_ULINT_TO_DINT, F_ULINT_TO_BYTE, F_WSTRING_TO_UDINT, F_TIME_TO_WSTRING, GET_STRUCT_VALUE, GEN_PUBLISH, F_REAL_TO_DWORD, F_DWORD_BCD_TO_UDINT, F_INT_TO_LREAL, F_SINT_TO_WSTRING, Conveyor1Check, F_LWORD_TO_SINT, F_GT, F_LINT_TO_REAL, F_TIME_IN_MS_TO_LINT, F_SINT_TO_REAL, F_LOG, F_ULINT_TO_INT, F_DWORD_TO_SINT, F_BOOL_TO_WORD, F_REAL_TO_USINT, E_SWITCH, F_LINT_TO_LREAL, F_STRING_TO_LINT, F_SINT_TO_USINT, F_DINT_TO_REAL, DINT2DINT, F_WORD_TO_ULINT, F_INT_TO_SINT, F_CONCAT_DATE_TOD, F_WSTRING_TO_LREAL, GET_AT_INDEX, F_USINT_TO_LREAL, F_BOOL_TO_WSTRING, FB_CTU_ULINT, F_DINT_TO_LREAL, UDINT2UDINT, F_USINT_TO_BYTE, F_BOOL_TO_STRING, F_LWORD_TO_DWORD, F_LREAL_TO_UDINT, F_STRING_TO_UDINT, F_UDINT_TO_DINT, F_UDINT_TO_BYTE, F_WSTRING_TO_LINT, F_USINT_TO_DINT)} (* created during deployment *)
    RESOURCE EMB_RES : EMB_RES
      FBS
        TransLeftCheck_1 : TransLeftCheck;
        Conveyor1Check : Conveyor1Check;
        Load1Check : Load1Check;
        AtEntry1 : SUBSCRIBE_1(QI := 1, ID := opc_ua[SUBSCRIBE;opc.tcp://localhost:4840#;/Objects/1:AtEntry1]);
        COnveyor1_Actuator : CLIENT_1_0(QI := 1, ID := opc_ua[WRITE;opc.tcp://localhost:4840#;/Objects/1:Conveyor1]);
        ExitCheck : ExitCheck;
        Load2Check : Load2Check;
        Conveyor2Check : Conveyor2Check;
        Load2_Acuator : CLIENT_1_0(QI := 1, ID := opc_ua[WRITE;opc.tcp://localhost:4840#;/Objects/1:Load2]);
        Reset : SUBSCRIBE_1(QI := 1, ID := opc_ua[SUBSCRIBE;opc.tcp://localhost:4840#;/Objects/1:Reset]);
        Load2 : SUBSCRIBE_1(QI := 1, ID := opc_ua[SUBSCRIBE;opc.tcp://localhost:4840#;/Objects/1:Load2]);
        TransLeft1 : SUBSCRIBE_1(QI := 1, ID := opc_ua[SUBSCRIBE;opc.tcp://localhost:4840#;/Objects/1:TransLeft1]);
        Load1 : SUBSCRIBE_1(QI := 1, ID := opc_ua[SUBSCRIBE;opc.tcp://localhost:4840#;/Objects/1:Load1]);
        TransLeft2 : SUBSCRIBE_1(QI := 1, ID := opc_ua[SUBSCRIBE;opc.tcp://localhost:4840#;/Objects/1:TransLeft2]);
        Conveyor2 : SUBSCRIBE_1(QI := 1, ID := opc_ua[SUBSCRIBE;opc.tcp://localhost:4840#;/Objects/1:Conveyor2]);
        ExitConv : SUBSCRIBE_1(QI := 1, ID := opc_ua[SUBSCRIBE;opc.tcp://localhost:4840#;/Objects/1:ExitConv]);
        E_DELAY : E_DELAY(DT := T#1s);
        AtTrans1 : SUBSCRIBE_1(QI := 1, ID := opc_ua[SUBSCRIBE;opc.tcp://localhost:4840#;/Objects/1:AtTrans1]);
        AtEntry2 : SUBSCRIBE_1(QI := 1, ID := opc_ua[SUBSCRIBE;opc.tcp://localhost:4840#;/Objects/1:AtEntry2]);
        Conveyor2_Actuator : CLIENT_1_0(QI := 1, ID := opc_ua[WRITE;opc.tcp://localhost:4840#;/Objects/1:Conveyor2]);
        AtTrans2 : SUBSCRIBE_1(QI := 1, ID := opc_ua[SUBSCRIBE;opc.tcp://localhost:4840#;/Objects/1:AtTrans2]);
        TransLeft2_Actuator : CLIENT_1_0(QI := 1, ID := opc_ua[WRITE;opc.tcp://localhost:4840#;/Objects/1:TransLeft2]);
        TransLeft1_Actuator : CLIENT_1_0(QI := 1, ID := opc_ua[WRITE;opc.tcp://localhost:4840#;/Objects/1:TransLeft1]);
        AtExit : SUBSCRIBE_1(QI := 1, ID := opc_ua[SUBSCRIBE;opc.tcp://localhost:4840#;/Objects/1:AtExit]);
        Start : SUBSCRIBE_1(QI := 1, ID := opc_ua[SUBSCRIBE;opc.tcp://localhost:4840#;/Objects/1:Start]);
        ExitConv_Acuator : CLIENT_1_0(QI := 1, ID := opc_ua[WRITE;opc.tcp://localhost:4840#;/Objects/1:ExitConv]);
        Load1_Actuator : CLIENT_1_0(QI := 1, ID := opc_ua[WRITE;opc.tcp://localhost:4840#;/Objects/1:Load1]);
        MyBasicTest : MyBasicTest;
      END_FBS
      EVENT_CONNECTIONS
        AtEntry1.IND TO TransLeftCheck_1.REQ;
        AtEntry1.IND TO Conveyor1Check.REQ;
        AtEntry1.IND TO Load1Check.REQ;
        Conveyor1Check.CNF TO COnveyor1_Actuator.REQ;
        Conveyor1Check.INITO TO COnveyor1_Actuator.INIT;
        Load2Check.CNF TO Load2_Acuator.REQ;
        TransLeft1.IND TO Conveyor1Check.REQ;
        TransLeft1.INITO TO Conveyor1Check.INIT;
        TransLeft2.IND TO Load2Check.REQ;
        TransLeft2.IND TO Load1Check.REQ;
        E_DELAY.EO TO AtEntry1.INIT;
        E_DELAY.EO TO Reset.INIT;
        E_DELAY.EO TO Load2.INIT;
        E_DELAY.EO TO TransLeft1.INIT;
        E_DELAY.EO TO Load1.INIT;
        E_DELAY.EO TO TransLeft2.INIT;
        E_DELAY.EO TO Conveyor2.INIT;
        E_DELAY.EO TO ExitConv.INIT;
        START.WARM TO E_DELAY.START;
        START.COLD TO E_DELAY.START;
        AtTrans1.IND TO TransLeftCheck_1.REQ;
        AtTrans1.IND TO Load1Check.REQ;
        E_DELAY.EO TO AtTrans1.INIT;
        AtEntry2.IND TO Load2Check.REQ;
        AtEntry2.INITO TO Load2_Acuator.INIT;
        E_DELAY.EO TO AtEntry2.INIT;
        Conveyor2Check.CNF TO Conveyor2_Actuator.REQ;
        AtTrans2.IND TO TransLeftCheck_1.REQ;
        AtTrans2.IND TO Conveyor2Check.REQ;
        AtTrans2.INITO TO Conveyor2_Actuator.INIT;
        E_DELAY.EO TO AtTrans2.INIT;
        TransLeftCheck_1.CNF TO TransLeft2_Actuator.REQ;
        AtTrans2.INITO TO TransLeft2_Actuator.INIT;
        TransLeftCheck_1.CNF TO TransLeft1_Actuator.REQ;
        AtTrans2.INITO TO TransLeft1_Actuator.INIT;
        AtExit.IND TO ExitCheck.REQ;
        E_DELAY.EO TO AtExit.INIT;
        E_DELAY.EO TO Start.INIT;
        ExitCheck.CNF TO ExitConv_Acuator.REQ;
        AtExit.INITO TO ExitConv_Acuator.INIT;
        Load1Check.CNF TO Load1_Actuator.REQ;
        AtTrans1.INITO TO Load1_Actuator.INIT;
        START.COLD TO MyBasicTest.INIT;
        START.WARM TO MyBasicTest.INIT;
      END_CONNECTIONS
      DATA_CONNECTIONS
        AtEntry1.RD_1 TO TransLeftCheck_1.AtEntry1;
        AtEntry1.RD_1 TO Conveyor1Check.AtEntry1;
        AtEntry1.RD_1 TO Load1Check.AtEntry1;
        Conveyor1Check.QO TO COnveyor1_Actuator.SD_1;
        Load2Check.QO TO Load2_Acuator.SD_1;
        TransLeft1.RD_1 TO Conveyor1Check.TransLeft;
        TransLeft2.RD_1 TO Load1Check.TransLeft;
        TransLeft2.RD_1 TO Load2Check.TransLeft2;
        AtTrans1.RD_1 TO TransLeftCheck_1.AtTrans1;
        AtTrans1.RD_1 TO Load1Check.AtTrans1;
        AtEntry2.RD_1 TO Load2Check.AtEntry2;
        Conveyor2Check.QO TO Conveyor2_Actuator.SD_1;
        AtTrans2.RD_1 TO TransLeftCheck_1.AtTrans2;
        AtTrans2.RD_1 TO Conveyor2Check.QI;
        TransLeftCheck_1.QO TO TransLeft2_Actuator.SD_1;
        TransLeftCheck_1.QO TO TransLeft1_Actuator.SD_1;
        AtExit.RD_1 TO ExitCheck.AtExit;
        ExitCheck.QO TO ExitConv_Acuator.SD_1;
        Load1Check.QO TO Load1_Actuator.SD_1;
      END_CONNECTIONS
    END_RESOURCE
  END_DEVICE
  MAPPINGS
    VariablesInitApp.E_DELAY ON FORTE_PC.EMB_RES.E_DELAY;
    VariablesInitApp.AtTrans2_Init ON FORTE_PC.EMB_RES.AtTrans2_Init;
    VariablesInitApp.AtExit_Init ON FORTE_PC.EMB_RES.AtExit_Init;
    VariablesInitApp.Load1_Init ON FORTE_PC.EMB_RES.Load1_Init;
    VariablesInitApp.ExitConv_Init ON FORTE_PC.EMB_RES.ExitConv_Init;
    VariablesInitApp.TransLeft2_Init ON FORTE_PC.EMB_RES.TransLeft2_Init;
    VariablesInitApp.AtTrans1_Init ON FORTE_PC.EMB_RES.AtTrans1_Init;
    VariablesInitApp.Reset_Init ON FORTE_PC.EMB_RES.Reset_Init;
    VariablesInitApp.Load2_Init ON FORTE_PC.EMB_RES.Load2_Init;
    VariablesInitApp.AtEntry2_Init ON FORTE_PC.EMB_RES.AtEntry2_Init;
    VariablesInitApp.Start_Init ON FORTE_PC.EMB_RES.Start_Init;
    VariablesInitApp.Conveyor2_Init ON FORTE_PC.EMB_RES.Conveyor2_Init;
    VariablesInitApp.TransLeft1_Init ON FORTE_PC.EMB_RES.TransLeft1_Init;
    VariablesInitApp.Conveyor1_Init ON FORTE_PC.EMB_RES.Conveyor1_Init;
    VariablesInitApp.AtEntry1_Init ON FORTE_PC.EMB_RES.AtEntry1_Init;
    VariablesInitApp.NodeInit ON FORTE_PC.EMB_RES.NodeInit;
    FactoryioLuaJITDemo.TransLeftCheck_1 ON FORTE_PC_1.EMB_RES.TransLeftCheck_1;
    FactoryioLuaJITDemo.Conveyor1Check ON FORTE_PC_1.EMB_RES.Conveyor1Check;
    FactoryioLuaJITDemo.Load1Check ON FORTE_PC_1.EMB_RES.Load1Check;
    FactoryioLuaJITDemo.AtEntry1 ON FORTE_PC_1.EMB_RES.AtEntry1;
    FactoryioLuaJITDemo.COnveyor1_Actuator ON FORTE_PC_1.EMB_RES.COnveyor1_Actuator;
    FactoryioLuaJITDemo.ExitCheck ON FORTE_PC_1.EMB_RES.ExitCheck;
    FactoryioLuaJITDemo.Load2Check ON FORTE_PC_1.EMB_RES.Load2Check;
    FactoryioLuaJITDemo.Conveyor2Check ON FORTE_PC_1.EMB_RES.Conveyor2Check;
    FactoryioLuaJITDemo.Load2_Acuator ON FORTE_PC_1.EMB_RES.Load2_Acuator;
    FactoryioLuaJITDemo.Reset ON FORTE_PC_1.EMB_RES.Reset;
    FactoryioLuaJITDemo.Load2 ON FORTE_PC_1.EMB_RES.Load2;
    FactoryioLuaJITDemo.TransLeft1 ON FORTE_PC_1.EMB_RES.TransLeft1;
    FactoryioLuaJITDemo.Load1 ON FORTE_PC_1.EMB_RES.Load1;
    FactoryioLuaJITDemo.TransLeft2 ON FORTE_PC_1.EMB_RES.TransLeft2;
    FactoryioLuaJITDemo.Conveyor2 ON FORTE_PC_1.EMB_RES.Conveyor2;
    FactoryioLuaJITDemo.ExitConv ON FORTE_PC_1.EMB_RES.ExitConv;
    FactoryioLuaJITDemo.E_DELAY ON FORTE_PC_1.EMB_RES.E_DELAY;
    FactoryioLuaJITDemo.AtTrans1 ON FORTE_PC_1.EMB_RES.AtTrans1;
    FactoryioLuaJITDemo.AtEntry2 ON FORTE_PC_1.EMB_RES.AtEntry2;
    FactoryioLuaJITDemo.Conveyor2_Actuator ON FORTE_PC_1.EMB_RES.Conveyor2_Actuator;
    FactoryioLuaJITDemo.AtTrans2 ON FORTE_PC_1.EMB_RES.AtTrans2;
    FactoryioLuaJITDemo.TransLeft2_Actuator ON FORTE_PC_1.EMB_RES.TransLeft2_Actuator;
    FactoryioLuaJITDemo.TransLeft1_Actuator ON FORTE_PC_1.EMB_RES.TransLeft1_Actuator;
    FactoryioLuaJITDemo.AtExit ON FORTE_PC_1.EMB_RES.AtExit;
    FactoryioLuaJITDemo.Start ON FORTE_PC_1.EMB_RES.Start;
    FactoryioLuaJITDemo.ExitConv_Acuator ON FORTE_PC_1.EMB_RES.ExitConv_Acuator;
    FactoryioLuaJITDemo.Load1_Actuator ON FORTE_PC_1.EMB_RES.Load1_Actuator;
    FactoryioLuaJITDemo.MyBasicTest ON FORTE_PC_1.EMB_RES.MyBasicTest;
  END_MAPPINGS
  SEGMENTS
    Ethernet : Ethernet;
  END_SEGMENTS
  LINKS
    FORTE_PC => Ethernet;
    FORTE_PC_1 => Ethernet;
  END_LINKS
END_SYSTEM
